INTERFACE PUBLIC ResettingCommands EXTENDS RunningStateCommands, ActionStateCommands

END_INTERFACE

(* stored: Version 1.1.0.1, ProductVersion 3.1.4026.18
   Itf ResettingCommands: Id {8d330c53-dd73-014c-3c2b-ac3d4e386b6d} *)
